FUNCTION_BLOCK FB_Axxe
VAR_INPUT
	i_i_AxxePosition	:	INT;
	i_i_AxxeMinPos		:	INT;
	i_i_AxxeMaxPos		:	INT;
END_VAR

METHOD M_SetAxxeValues : BOOL
VAR_INPUT
	AxxeMinPos		:	INT;
	AxxeMaxPos		:	INT;
END_VAR
i_i_AxxeMinPos:=AxxeMinPos;
i_i_AxxeMaxPos:=AxxeMaxPos;
IF i_i_AxxeMinPos = AxxeMinPos AND i_i_AxxeMaxPos = AxxeMaxPos THEN
	M_SetAxxeValues:=TRUE;	
END_IF
END_METHOD

END_FUNCTION_BLOCK

(* stored: Version 1.1.0.1, ProductVersion 3.1.4024.3
   POU FB_Axxe: Id {137564b9-828a-441c-a29e-142496d0fc9d}, SpecialFunc None
   Method M_SetAxxeValues: Id {307f6f91-7248-4993-a985-c29dd5090276} *)
